Xinje XDPPro project, PLC1: XD5-48-6Pls (software 3.5 2017-04-21)

PROGRAM Ladder

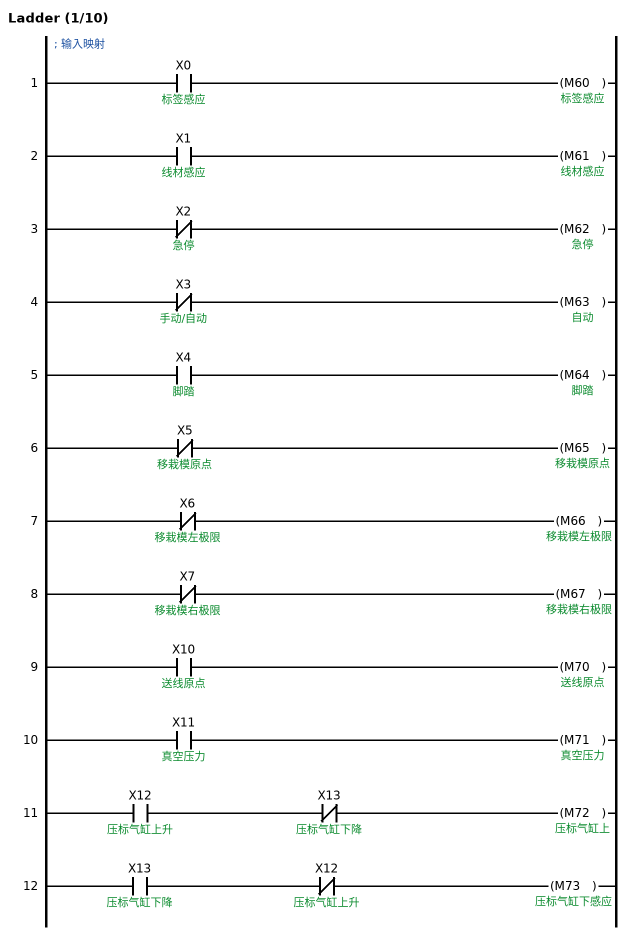
; 输入映射
LD     X0	; 标签感应
OUT    M60	; 标签感应
LD     X1	; 线材感应
OUT    M61	; 线材感应
LDI    X2	; 急停
OUT    M62	; 急停
LDI    X3	; 手动/自动
OUT    M63	; 自动
LD     X4	; 脚踏
OUT    M64	; 脚踏
LDI    X5	; 移栽模原点
OUT    M65	; 移栽模原点
LDI    X6	; 移栽模左极限
OUT    M66	; 移栽模左极限
LDI    X7	; 移栽模右极限
OUT    M67	; 移栽模右极限
LD     X10	; 送线原点
OUT    M70	; 送线原点
LD     X11	; 真空压力
OUT    M71	; 真空压力
LD     X12	; 压标气缸上升
ANI    X13	; 压标气缸下降
OUT    M72	; 压标气缸上
LD     X13	; 压标气缸下降
ANI    X12	; 压标气缸上升
OUT    M73	; 压标气缸下感应

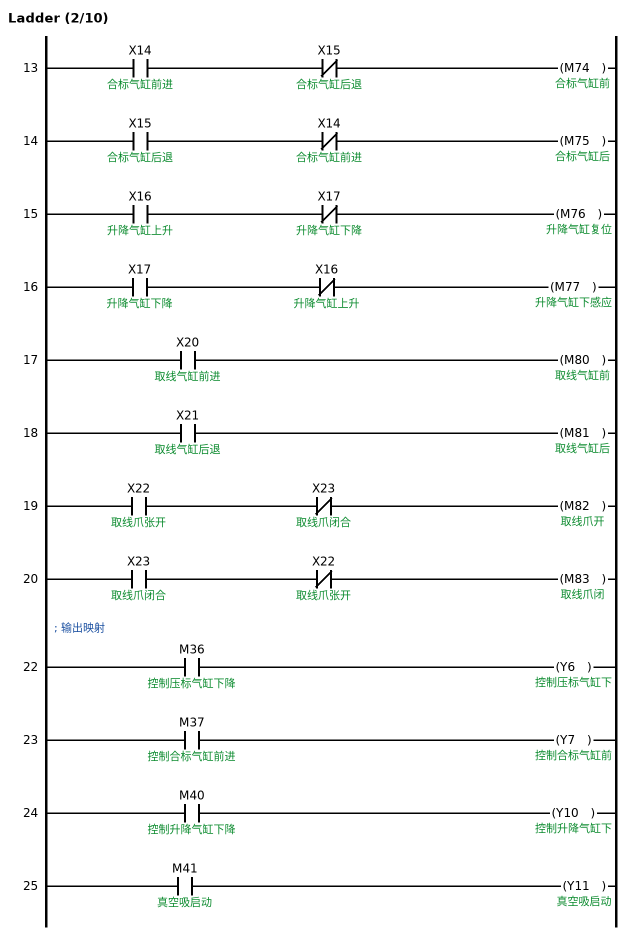
LD     X14	; 合标气缸前进
ANI    X15	; 合标气缸后退
OUT    M74	; 合标气缸前
LD     X15	; 合标气缸后退
ANI    X14	; 合标气缸前进
OUT    M75	; 合标气缸后
LD     X16	; 升降气缸上升
ANI    X17	; 升降气缸下降
OUT    M76	; 升降气缸复位
LD     X17	; 升降气缸下降
ANI    X16	; 升降气缸上升
OUT    M77	; 升降气缸下感应
LD     X20	; 取线气缸前进
OUT    M80	; 取线气缸前
LD     X21	; 取线气缸后退
OUT    M81	; 取线气缸后
LD     X22	; 取线爪张开
ANI    X23	; 取线爪闭合
OUT    M82	; 取线爪开
LD     X23	; 取线爪闭合
ANI    X22	; 取线爪张开
OUT    M83	; 取线爪闭
; 输出映射
LD     M36	; 控制压标气缸下降
OUT    Y6	; 控制压标气缸下
LD     M37	; 控制合标气缸前进
OUT    Y7	; 控制合标气缸前
LD     M40	; 控制升降气缸下降
OUT    Y10	; 控制升降气缸下
LD     M41	; 真空吸启动
OUT    Y11	; 真空吸启动

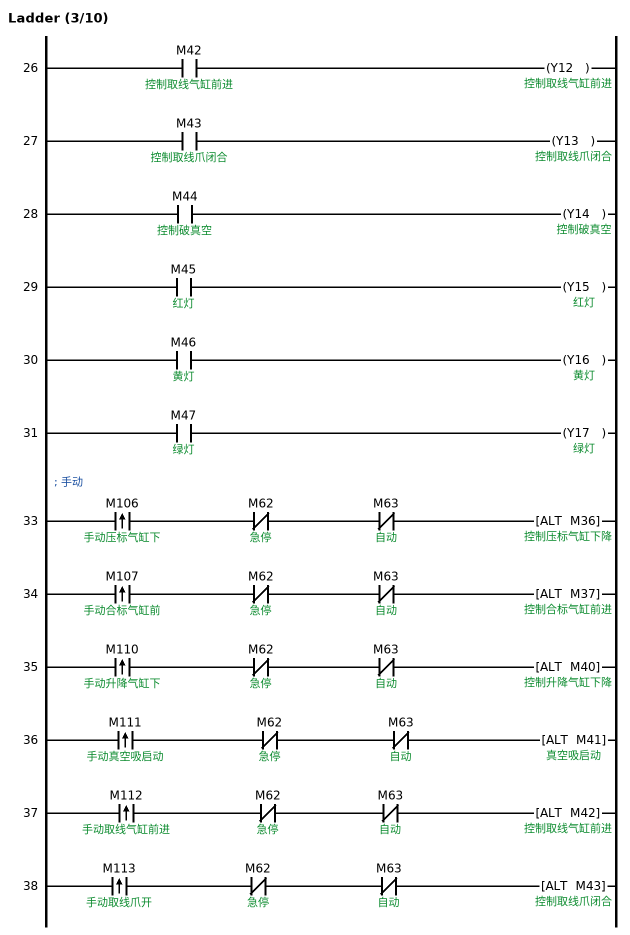
LD     M42	; 控制取线气缸前进
OUT    Y12	; 控制取线气缸前进
LD     M43	; 控制取线爪闭合
OUT    Y13	; 控制取线爪闭合
LD     M44	; 控制破真空
OUT    Y14	; 控制破真空
LD     M45	; 红灯
OUT    Y15	; 红灯
LD     M46	; 黄灯
OUT    Y16	; 黄灯
LD     M47	; 绿灯
OUT    Y17	; 绿灯
; 手动
LDP    M106	; 手动压标气缸下
ANI    M62	; 急停
ANI    M63	; 自动
ALT    M36	; 控制压标气缸下降
LDP    M107	; 手动合标气缸前
ANI    M62	; 急停
ANI    M63	; 自动
ALT    M37	; 控制合标气缸前进
LDP    M110	; 手动升降气缸下
ANI    M62	; 急停
ANI    M63	; 自动
ALT    M40	; 控制升降气缸下降
LDP    M111	; 手动真空吸启动
ANI    M62	; 急停
ANI    M63	; 自动
ALT    M41	; 真空吸启动
LDP    M112	; 手动取线气缸前进
ANI    M62	; 急停
ANI    M63	; 自动
ALT    M42	; 控制取线气缸前进
LDP    M113	; 手动取线爪开
ANI    M62	; 急停
ANI    M63	; 自动
ALT    M43	; 控制取线爪闭合

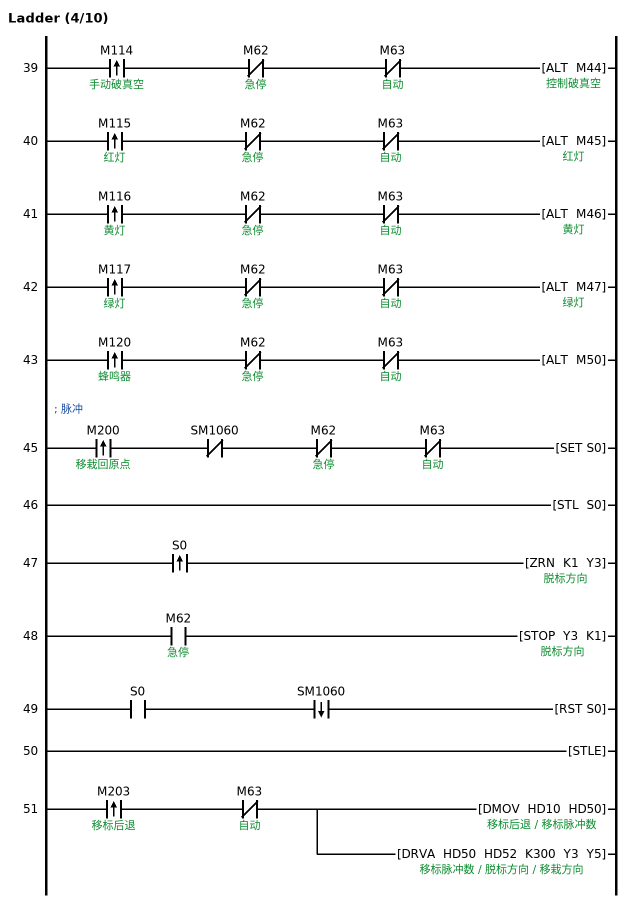
LDP    M114	; 手动破真空
ANI    M62	; 急停
ANI    M63	; 自动
ALT    M44	; 控制破真空
LDP    M115	; 红灯
ANI    M62	; 急停
ANI    M63	; 自动
ALT    M45	; 红灯
LDP    M116	; 黄灯
ANI    M62	; 急停
ANI    M63	; 自动
ALT    M46	; 黄灯
LDP    M117	; 绿灯
ANI    M62	; 急停
ANI    M63	; 自动
ALT    M47	; 绿灯
LDP    M120	; 蜂鸣器
ANI    M62	; 急停
ANI    M63	; 自动
ALT    M50
; 脉冲
LDP    M200	; 移栽回原点
ANI    SM1060
ANI    M62	; 急停
ANI    M63	; 自动
SET    S0
STL    S0
LDP    S0
ZRN    K1 Y3	; 脱标方向
LD     M62	; 急停
STOP   Y3 K1	; 脱标方向
LD     S0
ANDF   SM1060
RST    S0
STLE
LDP    M203	; 移标后退
ANI    M63	; 自动
DMOV   HD10 HD50	; 移标后退 / 移标脉冲数
DRVA   HD50 HD52 K300 Y3 Y5	; 移标脉冲数 / 脱标方向 / 移栽方向

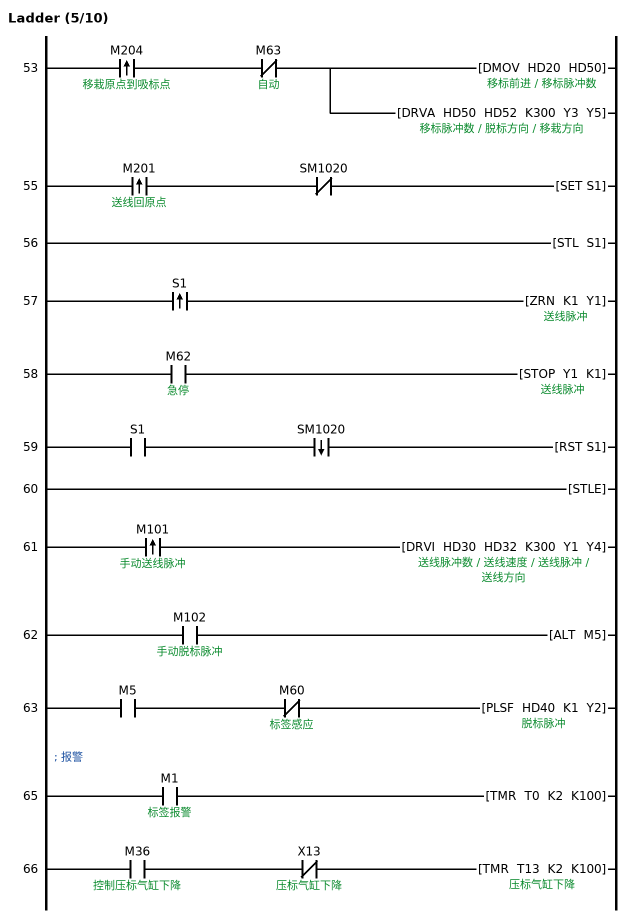
LDP    M204	; 移栽原点到吸标点
ANI    M63	; 自动
DMOV   HD20 HD50	; 移标前进 / 移标脉冲数
DRVA   HD50 HD52 K300 Y3 Y5	; 移标脉冲数 / 脱标方向 / 移栽方向
LDP    M201	; 送线回原点
ANI    SM1020
SET    S1
STL    S1
LDP    S1
ZRN    K1 Y1	; 送线脉冲
LD     M62	; 急停
STOP   Y1 K1	; 送线脉冲
LD     S1
ANDF   SM1020
RST    S1
STLE
LDP    M101	; 手动送线脉冲
DRVI   HD30 HD32 K300 Y1 Y4	; 送线脉冲数 / 送线速度 / 送线脉冲 / 送线方向
LD     M102	; 手动脱标脉冲
ALT    M5
LD     M5
ANI    M60	; 标签感应
PLSF   HD40 K1 Y2	; 脱标脉冲
; 报警
LD     M1	; 标签报警
TMR    T0 K2 K100
LD     M36	; 控制压标气缸下降
ANI    X13	; 压标气缸下降
TMR    T13 K2 K100	; 压标气缸下降

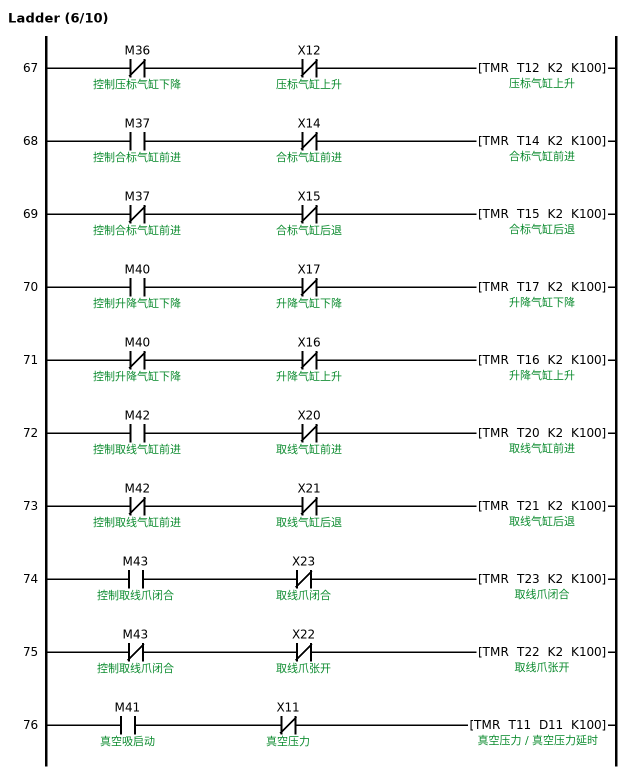
LDI    M36	; 控制压标气缸下降
ANI    X12	; 压标气缸上升
TMR    T12 K2 K100	; 压标气缸上升
LD     M37	; 控制合标气缸前进
ANI    X14	; 合标气缸前进
TMR    T14 K2 K100	; 合标气缸前进
LDI    M37	; 控制合标气缸前进
ANI    X15	; 合标气缸后退
TMR    T15 K2 K100	; 合标气缸后退
LD     M40	; 控制升降气缸下降
ANI    X17	; 升降气缸下降
TMR    T17 K2 K100	; 升降气缸下降
LDI    M40	; 控制升降气缸下降
ANI    X16	; 升降气缸上升
TMR    T16 K2 K100	; 升降气缸上升
LD     M42	; 控制取线气缸前进
ANI    X20	; 取线气缸前进
TMR    T20 K2 K100	; 取线气缸前进
LDI    M42	; 控制取线气缸前进
ANI    X21	; 取线气缸后退
TMR    T21 K2 K100	; 取线气缸后退
LD     M43	; 控制取线爪闭合
ANI    X23	; 取线爪闭合
TMR    T23 K2 K100	; 取线爪闭合
LDI    M43	; 控制取线爪闭合
ANI    X22	; 取线爪张开
TMR    T22 K2 K100	; 取线爪张开
LD     M41	; 真空吸启动
ANI    X11	; 真空压力
TMR    T11 D11 K100	; 真空压力 / 真空压力延时

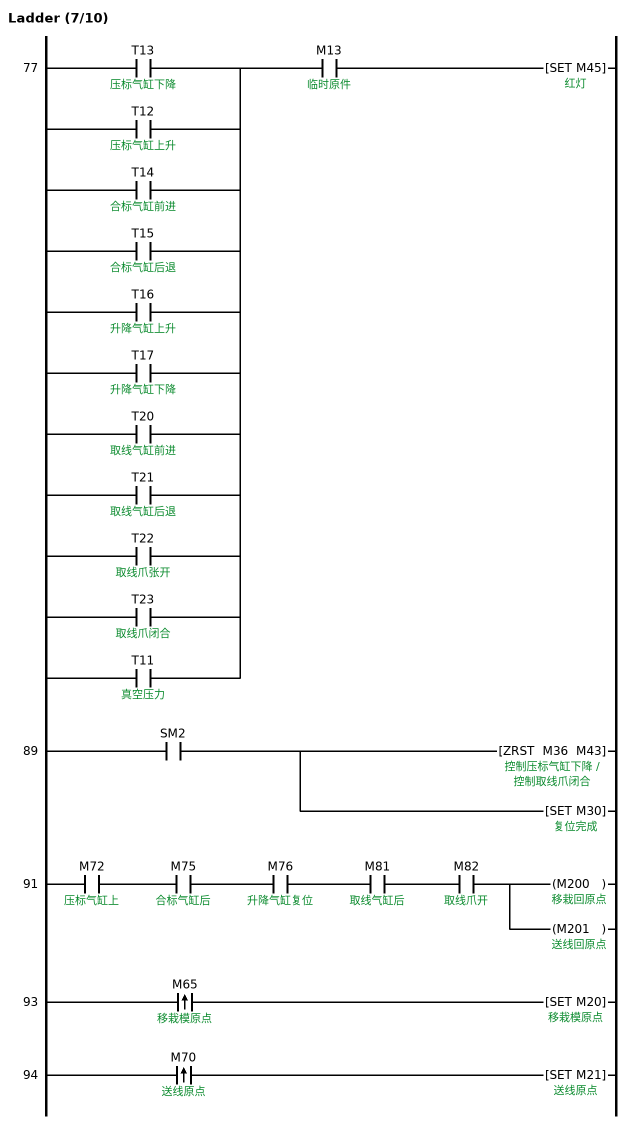
LD     T13	; 压标气缸下降
OR     T12	; 压标气缸上升
OR     T14	; 合标气缸前进
OR     T15	; 合标气缸后退
OR     T16	; 升降气缸上升
OR     T17	; 升降气缸下降
OR     T20	; 取线气缸前进
OR     T21	; 取线气缸后退
OR     T22	; 取线爪张开
OR     T23	; 取线爪闭合
OR     T11	; 真空压力
AND    M13	; 临时原件
SET    M45	; 红灯
LD     SM2
ZRST   M36 M43	; 控制压标气缸下降 / 控制取线爪闭合
SET    M30	; 复位完成
LD     M72	; 压标气缸上
AND    M75	; 合标气缸后
AND    M76	; 升降气缸复位
AND    M81	; 取线气缸后
AND    M82	; 取线爪开
OUT    M200	; 移栽回原点
OUT    M201	; 送线回原点
LDP    M65	; 移栽模原点
SET    M20	; 移栽模原点
LDP    M70	; 送线原点
SET    M21	; 送线原点

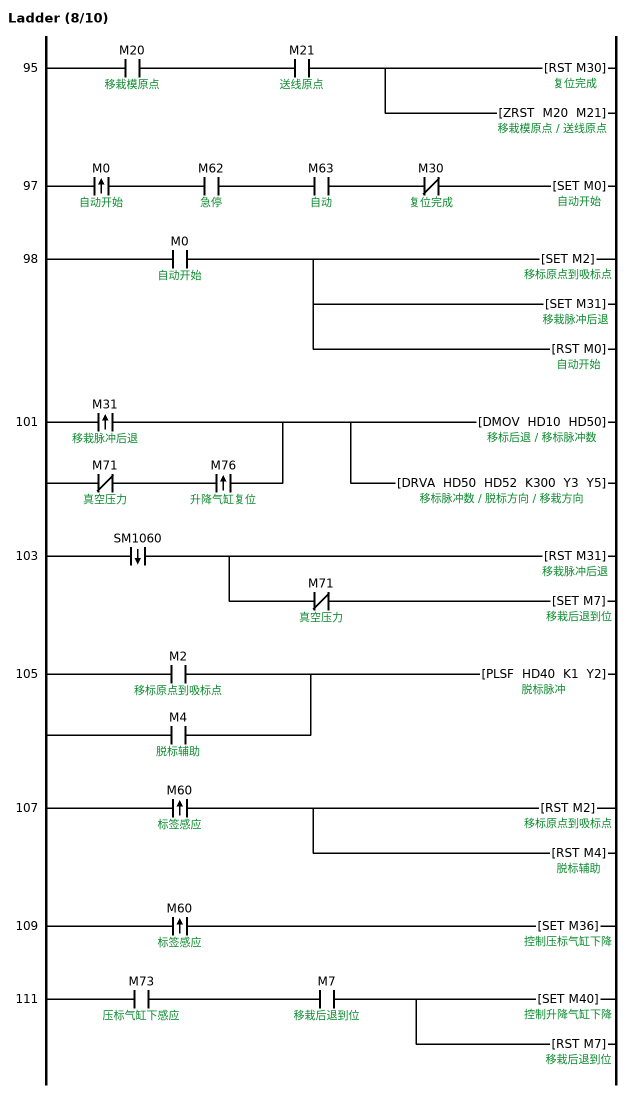
LD     M20	; 移栽模原点
AND    M21	; 送线原点
RST    M30	; 复位完成
ZRST   M20 M21	; 移栽模原点 / 送线原点
LDP    M0	; 自动开始
AND    M62	; 急停
AND    M63	; 自动
ANI    M30	; 复位完成
SET    M0	; 自动开始
LD     M0	; 自动开始
SET    M2	; 移标原点到吸标点
SET    M31	; 移栽脉冲后退
RST    M0	; 自动开始
LDP    M31	; 移栽脉冲后退
LDI    M71	; 真空压力
ANDP   M76	; 升降气缸复位
ORB
DMOV   HD10 HD50	; 移标后退 / 移标脉冲数
DRVA   HD50 HD52 K300 Y3 Y5	; 移标脉冲数 / 脱标方向 / 移栽方向
LDF    SM1060
RST    M31	; 移栽脉冲后退
ANI    M71	; 真空压力
SET    M7	; 移栽后退到位
LD     M2	; 移标原点到吸标点
OR     M4	; 脱标辅助
PLSF   HD40 K1 Y2	; 脱标脉冲
LDP    M60	; 标签感应
RST    M2	; 移标原点到吸标点
RST    M4	; 脱标辅助
LDP    M60	; 标签感应
SET    M36	; 控制压标气缸下降
LD     M73	; 压标气缸下感应
AND    M7	; 移栽后退到位
SET    M40	; 控制升降气缸下降
RST    M7	; 移栽后退到位

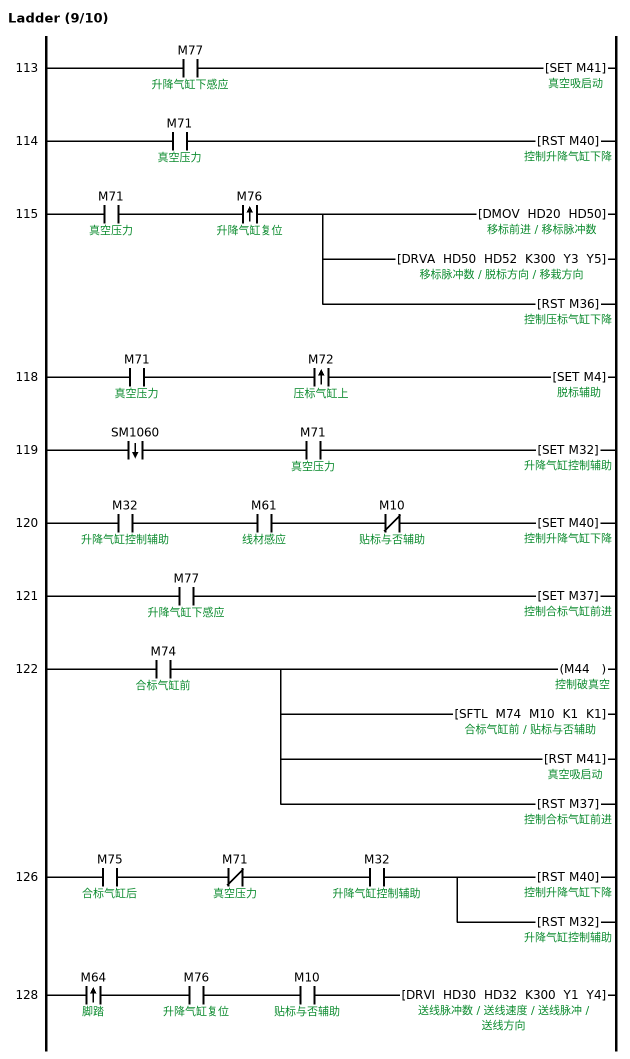
LD     M77	; 升降气缸下感应
SET    M41	; 真空吸启动
LD     M71	; 真空压力
RST    M40	; 控制升降气缸下降
LD     M71	; 真空压力
ANDP   M76	; 升降气缸复位
DMOV   HD20 HD50	; 移标前进 / 移标脉冲数
DRVA   HD50 HD52 K300 Y3 Y5	; 移标脉冲数 / 脱标方向 / 移栽方向
RST    M36	; 控制压标气缸下降
LD     M71	; 真空压力
ANDP   M72	; 压标气缸上
SET    M4	; 脱标辅助
LDF    SM1060
AND    M71	; 真空压力
SET    M32	; 升降气缸控制辅助
LD     M32	; 升降气缸控制辅助
AND    M61	; 线材感应
ANI    M10	; 贴标与否辅助
SET    M40	; 控制升降气缸下降
LD     M77	; 升降气缸下感应
SET    M37	; 控制合标气缸前进
LD     M74	; 合标气缸前
OUT    M44	; 控制破真空
SFTL   M74 M10 K1 K1	; 合标气缸前 / 贴标与否辅助
RST    M41	; 真空吸启动
RST    M37	; 控制合标气缸前进
LD     M75	; 合标气缸后
ANI    M71	; 真空压力
AND    M32	; 升降气缸控制辅助
RST    M40	; 控制升降气缸下降
RST    M32	; 升降气缸控制辅助
LDP    M64	; 脚踏
AND    M76	; 升降气缸复位
AND    M10	; 贴标与否辅助
DRVI   HD30 HD32 K300 Y1 Y4	; 送线脉冲数 / 送线速度 / 送线脉冲 / 送线方向

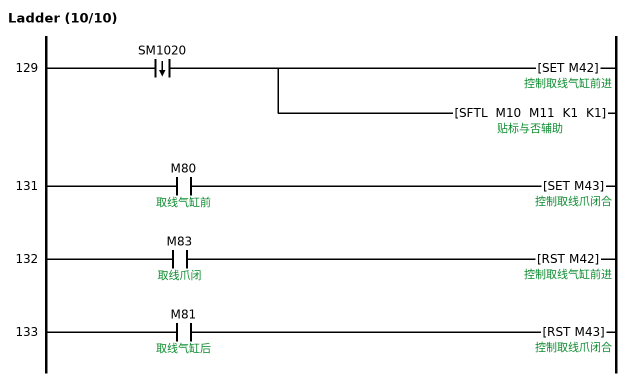
LDF    SM1020
SET    M42	; 控制取线气缸前进
SFTL   M10 M11 K1 K1	; 贴标与否辅助
LD     M80	; 取线气缸前
SET    M43	; 控制取线爪闭合
LD     M83	; 取线爪闭
RST    M42	; 控制取线气缸前进
LD     M81	; 取线气缸后
RST    M43	; 控制取线爪闭合

COMMENTS (devices not used above)
Y0	移栽脉冲
Y20	蜂鸣器
M3	压标气缸控制辅助
M6	送线定位
M33	真空吸控制辅助
M34	标签贴与否辅助
M100	手动移栽脉冲
M103	脱标方向
M104	送线方向
M105	移栽方向
M202	移标前进
M300	移标
HD0	移标前进